Staubli VAL3: processList.pjx

--- processList.pjx ---
Parameters version=s7.2.1 stackSize=5000 millimeterUnit=true
Program file=buildList.pgx
Program file=changeCycle.pgx
Program file=listAdd.pgx
Program file=loadPage.pgx
Program file=main.pgx
Program file=onEnterEvent.pgx
Program file=onExit.pgx
Program file=onF1Event.pgx
Program file=onF2Event.pgx
Program file=onF3Event.pgx
Program file=onF4Event.pgx
Program file=onF5Event.pgx
Program file=onF6Event.pgx
Program file=onF7Event.pgx
Program file=onF8Event.pgx
Program file=onLeftEvent.pgx
Program file=onRightEvent.pgx
Program file=onStart.pgx
Program file=programList.pgx
Program file=refresh.pgx
Program file=refreshDynamic.pgx
Program file=refreshStatic.pgx
Program file=selectType.pgx
Data file=processList.dtx
Library alias=saveData path=Disk://saveData/saveData.pjx
Library alias=use path=Disk://kernel/userPage/userPage.pjx
Library alias=cycleStatus path=Disk://cycleStatus/cycleStatus.pjx
Library alias=prog path=Disk://instruction/PROG/PROG.pjx
Library alias=page path=Disk://kernel/template/page/page.pjx
Library alias=language path=Disk://kernel/language/language.pjx
Library alias=processList path=Disk://kernel/processList/processList.pjx
Library alias=OnEvent path=Disk://OnEvent/OnEvent.pjx

--- processList.dtx ---
num nIndex
num nKey
num nRefresh
num nTime = 1
num nView
string sEvent
public string sItems
string sList
string sMenu[8]
string sMessage
string sType[3]
  [0] = "START Process"
  [1] = "MAIN Process"
  [2] = "END Process"
string sMenu8[8]
string sWrite
bool bButton[8]
bool bLarge

--- main.pgx ---
public program main()
begin
  // INIT
  call onStart()
  // LOOP UNTIL nKey=255
  do
    call refresh()
    nKey=getKey()
    call use:listevent(nKey,nIndex,sEvent)
    nView=use:nView
    switch nKey
      case 259
        // TAB
        bLarge=!bLarge
        call use:setView(bLarge)
      break
      case 264
        // left
        call onLeftEvent()
      break
      case 268
        // right
        call onRightEvent()
      break
      case 271
        call onF1Event()
      break
      case 272
        // set LOOP
        call onF2Event()
      break
      case 273
        call onF3Event()
      break
      case 274
        call onF4Event()
      break
      case 275
        call onF5Event()
      break
      case 276
        call onF6Event()
      break
      case 277
        // DELETE
        call onF7Event()
      break
      case 278
        // INSERT
        call onF8Event()
      break
      case 270
        // CHANGE THE NUMBER OF CYCLE
        call onEnterEvent()
      break
    endSwitch
    // release the resource
    delay(0)
  until nKey==255
  // on Exit
  call onExit()
end

--- buildList.pgx ---
program buildList()
  local num l_nSize
  local string l_sEvent
  local num i
  local string l_sProg
  local num l_nDone
  local num l_nTotal
  local num l_nType
  local string l_sItem
begin
  // INIT the list
  l_sItem=""
  call use:stringCopy(l_sItem,sList)
  // Build the list
  call processList:getDefaultType(l_nType)
  call processList:getSize(l_nSize,l_nType)
  if l_nSize>0
    for i=0 to (l_nSize-1)
      call processList:getCycle(l_sProg,l_nTotal,l_nDone,i,l_nType)
      if l_sProg!=""
        l_sEvent=(" ["+toString("1",l_nDone)+"/"+toString("1",l_nTotal)+"]")
        call listAdd(toString("2",i+1)+" "+l_sProg+l_sEvent)
      endIf
    endFor
  endIf
end

--- changeCycle.pgx ---
public program changeCycle(num x_nIndex, string x_sEvent)
  local num l_nSize
  local num l_nSwapTotal[3]
  local bool l_bCheck
  local num i
  local string l_sSwapProg[3]
  local num l_nTemp
  local num l_nTempTotal
  local string l_sProg
  local num l_sTotal
  local num l_nTempDone
  local num l_nType
  local string l_sEmpty
  local num l_nDone
  local num l_nZero
begin
  //
  //  copy the first 3 item of the processes' list,
  //  then l_bCheck if all it's OK
  //
  // check if the x_sEvent is not empty
  if x_sEvent!=""
    call processList:getDefaultType(l_nType)
    //for i=0 to 2
    call processList:getSize(l_nSize,l_nType)
    //endFor
    if l_nSize>2
      l_nSize=3
    endIf
    // make a backup of the first
    l_sEmpty=""
    l_nDone=0
    for i=0 to l_nSize-1
      call processList:getCycle(l_sSwapProg[i],l_nSwapTotal[i],l_nDone,i,l_nType)
    endFor
    // take the select one
    call processList:getCycle(l_sEmpty,l_nTempTotal,l_nDone,x_nIndex,l_nType)
    l_nTemp=l_nTempTotal
    //
    //  increase or Decrease the cicle to do1
    //
    i=find(x_sEvent,"/")
    // clean the line
    call use:listcursor(use:nView,false)
    l_sEmpty=""
    call use:changeValue(l_nTempTotal,1,999,i+40-use:nBottomX,x_nIndex+1,l_sEmpty)
    l_bCheck=false
    if l_nTempTotal!=l_nTemp
      for i=0 to l_nSize-1
        call processList:getCycle(l_sProg,l_sTotal,l_nDone,i,l_nType)
        if l_nSwapTotal[i]==l_sTotal and l_sSwapProg[i]==l_sProg
          l_bCheck=true
        endIf
      endFor
    endIf
    //
    // Check if the robot has the same processes' list
    //
    if l_bCheck
      //
      //  Change the totalcycle only if it is mayor then the doneCycle
      //
      l_nZero=0
      call processList:getCycle(l_sProg,l_nZero,l_nTempDone,x_nIndex,l_nType)
      if l_nTempTotal!=l_nTemp and l_nTempTotal>l_nTempDone
        call processList:setCycle(l_sProg,l_nTempTotal,l_nTempDone,x_nIndex,l_nType)
      endIf
    endIf
  endIf
end

--- listAdd.pgx ---
program listAdd(string x_sEvent)
begin
  // add in the queue not maintenane prog
  if sList!=""
    insert(sList[size(sList)])
  endIf
  sList[size(sList)-1]=x_sEvent
end

--- loadPage.pgx ---
program loadPage(string x_sPage, string& x_sItems[])
// load the next page
  local num i
  local string l_sMessage
begin
  // look if the page libload is correct
  i=page:libLoad(x_sPage)
  delay(0)
  if i!=0
    logMsg("[KERNEL] INTERFACE:PAGE LIBLOAD "+x_sPage+" result "+toString("",i))
    call language:message(l_sMessage,-7)
    popUpMsg(l_sMessage+x_sPage+" ; "+toString("",i))
  else
    // copy all the field from x_sItems to the next page
    call use:stringCopy(x_sItems,page:sItems)
    call page:main()
    // to give back
    call use:stringCopy(page:sItems,x_sItems)
  endIf
end

--- onEnterEvent.pgx ---
program onEnterEvent()
begin
  //
  // NB sEvent is the selected
  // element in the LIST
  //
  //
  // Change the cycle to do
  //
  if sEvent!=""
    call changeCycle(nIndex,sEvent)
    // logMsg
    logMsg("[KERNEL] CYCLEKEYEVENT:Change cycle to do for the program: "+sEvent+" at position: "+toString("",nIndex))
  endIf
end

--- onExit.pgx ---
program onExit()
begin
  // save the process list
  call processList:save()
  logMsg("[KERNEL] INTERFACE:Save process list")
end

--- onF1Event.pgx ---
program onF1Event()
  local bool l_bLoop
begin
  // look if the bButton is enable
  if bButton[0]
    //
    //  Set the LOOP ON/OFF
    //
    logMsg("[KERNEL] INTERFACE:Change the loop status")
    call processList:getLoop(l_bLoop)
    call processList:setLoop(!l_bLoop)
  endIf
end

--- onF2Event.pgx ---
program onF2Event()
  local num l_nSize[3]
  local string l_sEvent
  local num i
  local string l_sProg
  local num l_nDone
  local num l_nTotal
  local num l_nType
  local bool l_bLoop
  local num l_sType
  local string l_sEmpty
  local string l_sMessage
begin
  do
    cls()
    call language:message(l_sMessage,76)
    title("< "+l_sMessage+" >")
    call use:setView(true)
    // INIT the list
    l_sEmpty=""
    call use:stringCopy(l_sEmpty,sList)
    // get the LOOP
    call processList:getLoop(l_bLoop)
    // Build the list
    for i=0 to 2
      call processList:getSize(l_nSize[i],i)
    endFor
    //
    for l_nType=0 to 2
      switch l_nType
        case 0
          // START LIST
          call language:message(l_sMessage,72)
          l_sEmpty=(" "+l_sMessage)
          call use:strfill(l_sEmpty,17,l_sEmpty)
          l_sEmpty=l_sEmpty+":"
        break
        case 1
          call listAdd(" ")
          call language:message(l_sMessage,73)
          l_sEmpty=(" "+l_sMessage)
          call use:strfill(l_sEmpty,17,l_sEmpty)
          l_sEmpty=l_sEmpty+":"
          call processList:getLoop(l_bLoop)
        break
        case 2
          call listAdd(" ")
          call language:message(l_sMessage,74)
          l_sEmpty=(" "+l_sMessage)
          call use:strfill(l_sEmpty,17,l_sEmpty)
          l_sEmpty=l_sEmpty+":"
        break
      endSwitch
      //
      if l_nSize[l_nType]>0
        for i=0 to (l_nSize[l_nType]-1)
          if i!=0
            call use:strfill("",17,l_sEmpty)
          endIf
          // get the info
          call processList:getCycle(l_sProg,l_nTotal,l_nDone,i,l_nType)
          // if exist
          if l_sProg!=""
            // cycle done
            l_sEvent=(" "+toString("1",l_nDone)+"/"+toString("1",l_nTotal))
            if l_nType!=1 or !l_bLoop
              call listAdd(l_sEmpty+"   "+l_sProg+l_sEvent)
            else
              if l_nSize[1]==1
                call listAdd(l_sEmpty+"@> "+l_sProg+l_sEvent)
              else
                if i==0
                  call listAdd(l_sEmpty+"┌> "+l_sProg+l_sEvent)
                else
                  if i!=(l_nSize[l_nType]-1)
                    call listAdd(l_sEmpty+"││ "+l_sProg+l_sEvent)
                  else
                    call listAdd(l_sEmpty+"└┘ "+l_sProg+l_sEvent)
                  endIf
                endIf
              endIf
            endIf
          else
            // ONLY THE TAG
            call listAdd(l_sEmpty)
          endIf
        endFor
      endIf
    endFor
    // BUILD LIST
    call use:listcreate("")
    call use:listadd(sList)
    call use:listupdate(0)
    call language:message(l_sMessage,75)
    call use:type(40-getDisplayLen(l_sMessage),13,l_sMessage)
    //
    //
    do
      nKey=get()
      call use:listevent(nKey,nIndex,sEvent)
      if nKey==278
        for i=0 to 2
          call processList:deleteAll(i)
          // TO DO END CYCLE?
        endFor
      endIf
    until nKey==278 or nKey==255
  until nKey==255
  // refresh
  use:bUseRefresh=true
  call use:nullKey(nKey)
end

--- onF3Event.pgx ---
program onF3Event()
  local num i
  local num l_nSize[3]
  local num l_nType
  local string l_sProg
  local string l_sFill
  local num j
begin
  // look if the bButton is enable
  if bButton[2]
    // generate the file of the production
    call processList:makeFile()
  endIf
end

--- onF5Event.pgx ---
program onF5Event()
begin
  // look if the bButton is enable
  if bButton[4]
    //
    call selectType()
  endIf
end

--- onF6Event.pgx ---
program onF6Event()
  local string l_sMessage
  local num l_nType
begin
  // look if the bButton is enable
  if bButton[5]
    //
    //  Clear all the List
    //
    call processList:getDefaultType(l_nType)
    logMsg("[KERNEL] INTERFACE:Clear the list")
    call processList:deleteAll(l_nType)
    if cycleStatus:bCycle
      call language:message(l_sMessage,3)
      popUpMsg(l_sMessage)
    endIf
    sEvent=""
    nIndex=0
  endIf
end

--- onF7Event.pgx ---
program onF7Event()
  local string l_sMessage
  local num l_nType
begin
  // look if the bButton is enable
  if bButton[6]
    //
    //  Delete the selected process
    //
    call processList:getDefaultType(l_nType)
    call processList:delete(nIndex,l_nType)
    logMsg("[KERNEL] INTERFACE:Delete the program: "+sEvent+" at the index: "+toString("",nIndex))
    if nIndex==0 and cycleStatus:bCycle
      call OnEvent:endCycle()
      call language:message(l_sMessage,3)
      popUpMsg(l_sMessage)
    endIf
  endIf
end

--- onF8Event.pgx ---
program onF8Event()
  local string l_sProgram
  local string l_sMessage
  local num l_nTotal
  local num l_nType
  local num l_nZero
begin
  // look if the bButton is enable
  if bButton[7]
    //
    //  Insert a new program in the processes' List
    //
    call processList:getDefaultType(l_nType)
    l_nZero=0
    call processList:getCycle(l_sProgram,l_nZero,l_nZero,l_nZero,l_nType)
    if nIndex<=0 and l_sProgram=="" or sEvent==""
      nIndex=0
    else
      nIndex=nIndex+1
    endIf
    // list of the program
    call programList(l_sProgram)
    if l_sProgram!=""
      call language:message(l_sMessage,27)
      l_nTotal=1
      call use:insertDialog(l_sMessage+"##"+l_sProgram,l_nTotal,1,999)
      if !use:bUseEscape
        call processList:insertCycle(nIndex,l_sProgram,l_nTotal,0,l_nType)
        logMsg("[KERNEL] CYCLEKEYEVENT:Insert the new program: "+l_sProgram)
      endIf
    endIf
  endIf
end

--- onLeftEvent.pgx ---
program onLeftEvent()
  local num l_nDefault
  local num l_nSize
begin
  l_nSize=3
  // step -1
  call processList:getDefaultType(l_nDefault)
  l_nDefault=(l_nDefault+2)%(l_nSize)
  call processList:setDefaultType(l_nDefault)
  use:bUseRefresh=true
end

--- onRightEvent.pgx ---
program onRightEvent()
  local num l_nDefault
  local num l_nSize
begin
  l_nSize=3
  // step -1
  call processList:getDefaultType(l_nDefault)
  l_nDefault=(l_nDefault+1)%(l_nSize)
  call processList:setDefaultType(l_nDefault)
  use:bUseRefresh=true
end

--- onStart.pgx ---
program onStart()
  local num i
begin
  // logMsg
  logMsg("[KERNEL] INTERFACE:PAGE Process List")
  // reset the Key pressure
  call use:nullKey(nKey)
  // define the list
  call buildList()
  // build the page
  call refreshStatic()
  //
end

--- programList.pgx ---
program programList(string& x_sEvent[])
  local num nSize
  local string sEvent
  local num lKey
  local num i
  local string message
begin
  //
  // USE this procedure to view Prog
  // that you have already saved
  //
  cls()
  call use:setView(false)
  //
  // Prog
  //
  call use:listcreate("PROG ")
  //
  call prog:getSize(nSize)
  // refresh the list
  for i=0 to nSize-1
    call prog:get(sEvent,i)
    if sEvent!="" and find(sEvent,"#")==-1 and sEvent!="HOME1" and sEvent!="HOME2"
      call use:listadd(sEvent)
    endIf
  endFor
  call use:listupdate(0)
  call language:message(message,60)
  call use:typeLen(0,13,message,40)
  do
    lKey=get()
    call use:listevent(lKey,i,x_sEvent)
  until lKey==270 or lKey==255
  if lKey==255
    x_sEvent=""
  endIf
end

--- refresh.pgx ---
program refresh()
// // page refresh
begin
  // refresh the static message
  if (nKey>=270 and nKey<=278) or use:bUseRefresh
    call refreshStatic()
    call refreshDynamic()
  else
    // refresh the Dynamic message
    if abs(clock()-nRefresh)>nTime
      call refreshDynamic()
    endIf
  endIf
end

--- refreshDynamic.pgx ---
program refreshDynamic()
begin
  // DO NOT CHANGE
  nRefresh=clock()
  use:bUseRefresh=false
  //
  // ADD HERE
  //
  // build the list
  call buildList()
  call use:listempty()
  call use:listadd(sList)
  //
  //
  // refresh the cursor
  use:nView=nView
  // refresh the list
  call use:listupdate(0)
end

--- refreshStatic.pgx ---
program refreshStatic()
  local string l_sMenu
  local string l_sMessage
  local num l_nType
  local bool l_bLoop
begin
  cls()
  //
  // set the view of the page..
  //
  // SET THE PAGE NUMBER
  use:nPage=1020
  // USE <>PROFILE for <>PAGE
  use:nPage=use:nPage+abs(limit(saveData:mode,0,2)-2)
    // load the menu page
  if saveData:language!="japanese"
    // SET THE VIEW OF THE PAGE
    call language:page(l_sMessage,use:nPage)
    // define the menu
    call use:stringToArray(l_sMessage,sMenu)
  else
    // japanese use the array for the menu
    call language:page(sMenu8,use:nPage)
    call use:stringCopy(sMenu8,sMenu)
  endIf
  //
  // LOOP OR NO LOOP
  call processList:getDefaultType(l_nType)
  if l_nType!=1
    sMenu=""
  endIf
  if saveData:language!="japanese"
    // set the menu
    call use:setMenu(sMenu,true,3)
  else
    call use:setMenu(sMenu,false,3)
  endIf
  call use:getMenu(sMenu,bButton)
  //
  //  LOOP MODE only on Process List
  //
  if l_nType==1
    call processList:getLoop(l_bLoop)
    if l_bLoop
      call use:type(9,3,"->ON ")
    else
      call use:type(9,3,"->OFF")
    endIf
  endIf
  //
  // CREATE THE LIST
  //
  // define your list size for default
  call use:setSizeList(19,0,19,11)
  call use:setView(false)
  call use:listcreate(sType[l_nType])
  //
end

--- selectType.pgx ---
program selectType()
  local string l_sMessage
  local num l_nIndex
  local string l_sEvent
  local num l_nDefault
  local num l_nKey
  local num i
begin
  // change the processList
  call use:clear(0,13)
  call language:message(l_sMessage,191)
  call use:typeCenter(13,l_sMessage,40,true)
  call use:setSizeList(10,2,15,6)
  // build the list
  call use:listcreate(sMenu[4])
  call use:listadd(sType)
  call processList:getDefaultType(l_nDefault)
  call use:selectNewField(l_nDefault,0,0)
  // select the Item
  do
    l_nKey=get()
    call use:listevent(l_nKey,l_nIndex,l_sEvent)
  until l_nKey==270 or l_nKey==255
  if l_nKey==270
    call processList:setDefaultType(l_nIndex)
    use:bUseRefresh=true
  endIf
  //
end
